// TIA Portal V18 export
FUNCTION_BLOCK "__mot_universal_"   // FB18, FBD
{ S7_Optimized_Access := 'TRUE' }
VERSION : 0.1
// stored: AutoNumber true, IsIECCheckEnabled false, IsRetainMemResEnabled false, MemoryReserve 100, SetENOAutomatically false, UDAEnableTagReadback false
   VAR_INPUT
      ALLOWED : Bool;
      ALLOWED_ONLY_IN_OVERRIDE : Bool;
      OVERRIDE_NOW : Bool;
      isMultiturn : Bool;
      MultiTurnGoesFwdOnly : Bool;
      xFwdOk : Bool;
      xRevOk : Bool;
      xPredefCal : Bool;
      MAN_SET_SPEED_maxParSpeed : Real;
      ENC : Real;
      par : "typeMotPara";
      partnerCalibrated : Bool := true;
      artLimits : Bool;
      artLimFwd : Real;
      artLimRev : Real;
      AU_EXECUTE_TO_TARGET : Bool;
      AU_SPD : Real;
      AUT_MD_SPD_notPos : Bool := false;
      AUT : Bool;
      MAN : Bool;
      CLOCK_S_P_SCAN { ExternalWritable := 'False'} : Real;
      ALIEN_HOST_CONTROL_MODE_ENABLE : Bool;
      ALIEN_FWD : Bool;
      ALIEN_REV : Bool;
      ALIEN_SPEED_ABS : Real;
      TheseAreDoors : Bool;
   END_VAR
   VAR_OUTPUT
      AU_INPOS : Bool;
      FWD : Bool;
      REV : Bool;
      BRK_REL : Bool;
      SPEED_ABS : Real;
      SPEED : Real;
      BLIND : Bool;
      ER_FOLLOW : Bool;
      ER_SET : Bool;
      ER_FWD : Bool;
      ER_REV : Bool;
      er_ws : WString;
   END_VAR
   VAR_IN_OUT
      AU_TRGT : Real;
      calibrated : Bool;
      POS : Real;
      ENC_RET_DATA : "typePOSMEMcalib";
   END_VAR
   VAR
      par_Local : "typeMotPara";
      SERV_block : Bool;
      AUTO_static : Bool;
      MAN_static : Bool := TRUE;
      M_MD { S7_SetPoint := 'True'} : "MD";
      ENC_DB { S7_SetPoint := 'True'} : "encoder";
      manual { S7_SetPoint := 'True'} : "manual_analog";
      auto { S7_SetPoint := 'True'} : "auto_analog_NORMAL";
      ENC_CHECK { S7_SetPoint := 'True'} : "enc_no_change_in_time";
      BRK_DB { S7_SetPoint := 'True'} : "BRK_FB";
      sr_auto { S7_SetPoint := 'True'} : "SR_TRIG";
      sr_man { S7_SetPoint := 'True'} : "SR_TRIG";
      auto_analog_Speed_Instance { S7_SetPoint := 'True'} : "auto_analog_copySpeed";
      speed_slowed_by_inertia : Real;
      speed_command : Real;
      mot_speed_wdir_slowly_accelerated_Instance { S7_SetPoint := 'True'} : "mot_speed_wdir_slowly_accelerated";
      mot_missed_target { S7_SetPoint := 'True'} : "mot_universal_arrived_missed";
      arrived_missed : Bool;
   END_VAR
   VAR_TEMP
      reset_y : Bool;
      BRK_NOW_ERROR_EXISTS : Bool;
      speed_fast_neg : Real;
      placeHolderreal : Real;
      er_set_1m : Bool;
      er_set_1a1 : Bool;
      er_set_1a2 : Bool;
      er_set_2 : Bool;
      er_set_3 : Bool;
      inertia_Mode : Bool;
      erws1m0 : WString;
      erws1a1 : WString;
      erws1a2 : WString;
      erws2 : WString;
      erws3 : WString;
   END_VAR
   VAR CONSTANT
      erwsNOER : WString := WSTRING#'no er';
   END_VAR
BEGIN

REGION Network 1
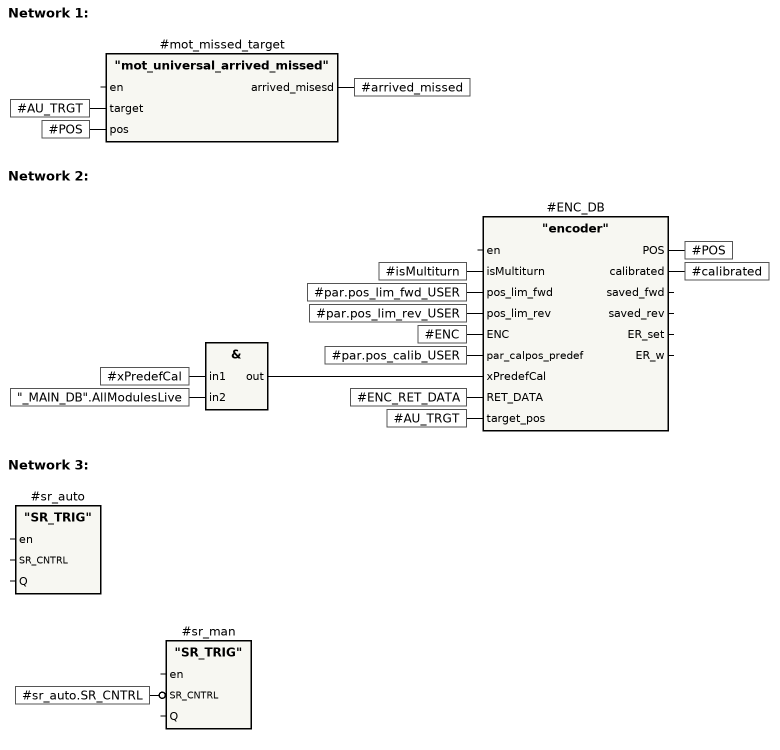
   #mot_missed_target(target := #AU_TRGT, pos := #POS, arrived_misesd => #arrived_missed);   // "mot_universal_arrived_missed"
END_REGION

REGION Network 2
   #ENC_DB(isMultiturn := #isMultiturn,   // "encoder"
           pos_lim_fwd := #par.pos_lim_fwd_USER,
           pos_lim_rev := #par.pos_lim_rev_USER,
           ENC := #ENC,
           par_calpos_predef := #par.pos_calib_USER,
           xPredefCal := #xPredefCal AND "_MAIN_DB".AllModulesLive,
           RET_DATA := #ENC_RET_DATA,
           target_pos := #AU_TRGT,
           POS => #POS,
           calibrated => #calibrated);
END_REGION

REGION Network 3
   #sr_auto();   // "SR_TRIG"
   #sr_man(SR_CNTRL := NOT #sr_auto.SR_CNTRL);   // "SR_TRIG"
END_REGION

REGION Network 4 (SCL)
   #SERV_block := #ALIEN_HOST_CONTROL_MODE_ENABLE;
   IF #SERV_block THEN
       #FWD := #ALIEN_FWD;
       #REV := #ALIEN_REV;
       #SPEED_ABS := #ALIEN_SPEED_ABS;
   END_IF;
END_REGION

REGION Network 5
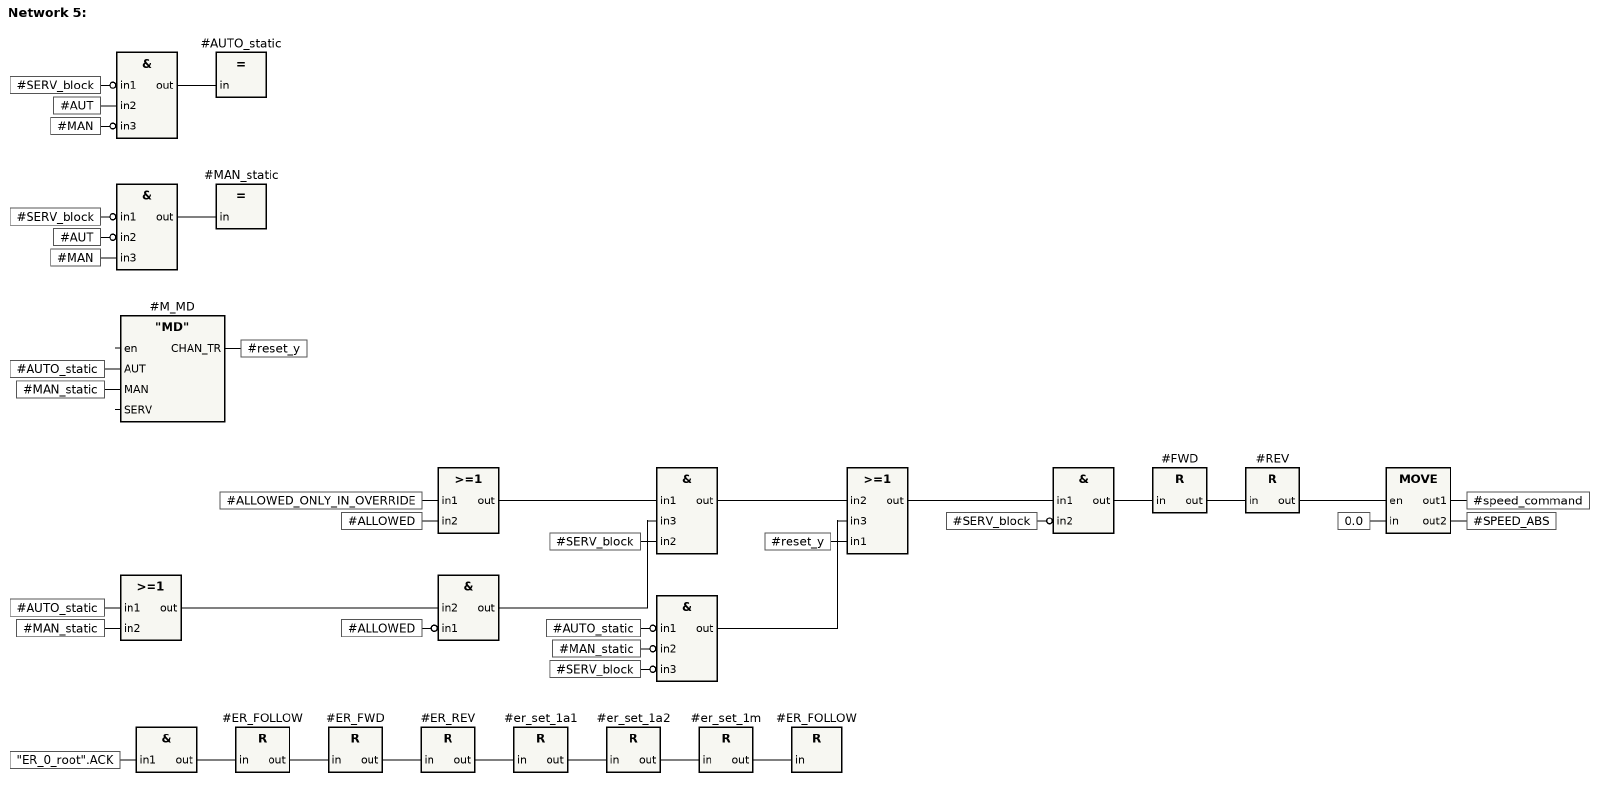
   #AUTO_static := NOT #SERV_block AND #AUT AND NOT #MAN;
   #MAN_static := NOT #SERV_block AND NOT #AUT AND #MAN;
   #M_MD(AUT := #AUTO_static, MAN := #MAN_static, CHAN_TR => #reset_y);   // "MD"
   IF (((#ALLOWED_ONLY_IN_OVERRIDE OR #ALLOWED) AND (#AUTO_static OR #MAN_static) AND NOT #ALLOWED AND #SERV_block) OR (NOT #AUTO_static AND NOT #MAN_static AND NOT #SERV_block) OR #reset_y) AND NOT #SERV_block THEN
       #FWD := FALSE;
       #REV := FALSE;
       #speed_command := 0.0;
       #SPEED_ABS := 0.0;
   END_IF;
   IF "ER_0_root".ACK THEN
       #ER_FOLLOW := FALSE;
       #ER_FWD := FALSE;
       #ER_REV := FALSE;
       #er_set_1a1 := FALSE;
       #er_set_1a2 := FALSE;
       #er_set_1m := FALSE;
       #ER_FOLLOW := FALSE;
   END_IF;
END_REGION

REGION Network 6
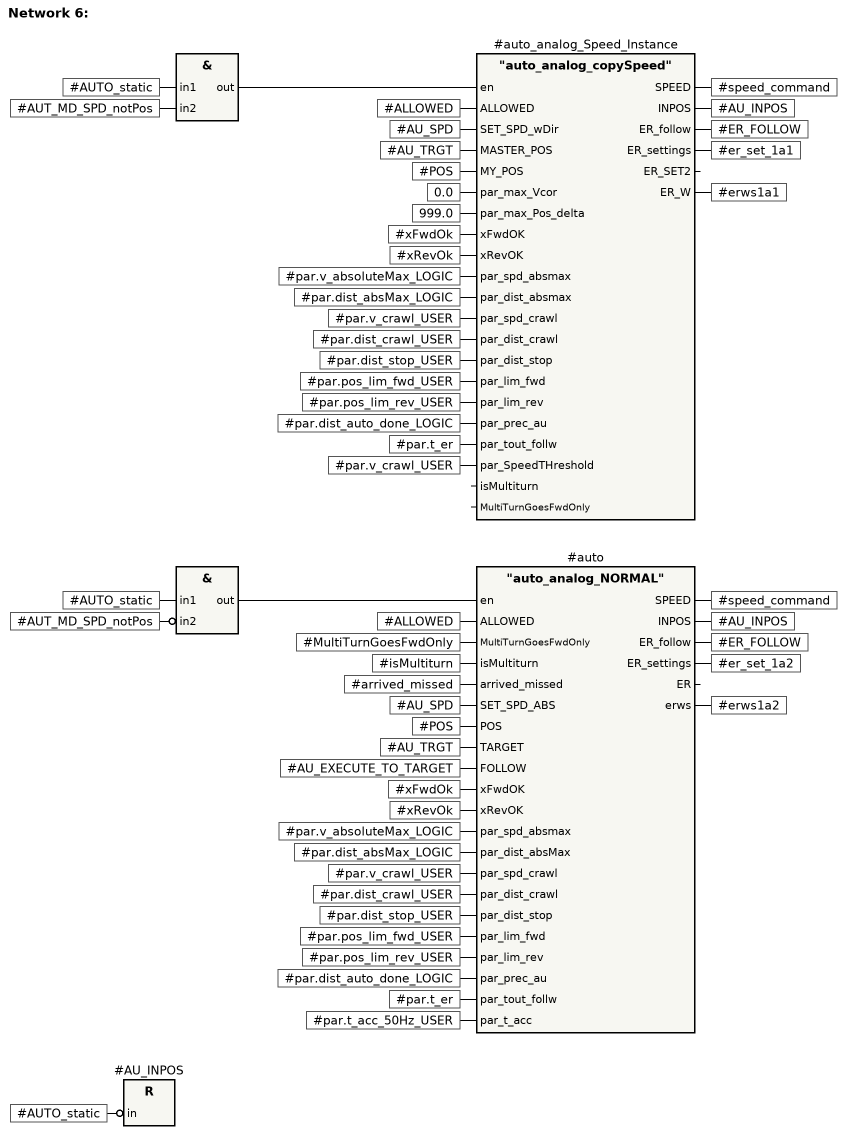
   IF #AUTO_static AND #AUT_MD_SPD_notPos THEN
       #auto_analog_Speed_Instance(ALLOWED := #ALLOWED,   // "auto_analog_copySpeed"
                               SET_SPD_wDir := #AU_SPD,
                               MASTER_POS := #AU_TRGT,
                               MY_POS := #POS,
                               par_max_Vcor := 0.0,
                               par_max_Pos_delta := 999.0,
                               xFwdOK := #xFwdOk,
                               xRevOK := #xRevOk,
                               par_spd_absmax := #par.v_absoluteMax_LOGIC,
                               par_dist_absmax := #par.dist_absMax_LOGIC,
                               par_spd_crawl := #par.v_crawl_USER,
                               par_dist_crawl := #par.dist_crawl_USER,
                               par_dist_stop := #par.dist_stop_USER,
                               par_lim_fwd := #par.pos_lim_fwd_USER,
                               par_lim_rev := #par.pos_lim_rev_USER,
                               par_prec_au := #par.dist_auto_done_LOGIC,
                               par_tout_follw := #par.t_er,
                               par_SpeedTHreshold := #par.v_crawl_USER,
                               SPEED => #speed_command,
                               INPOS => #AU_INPOS,
                               ER_follow => #ER_FOLLOW,
                               ER_settings => #er_set_1a1,
                               ER_W => #erws1a1);
   END_IF;
   IF #AUTO_static AND NOT #AUT_MD_SPD_notPos THEN
       #auto(ALLOWED := #ALLOWED,   // "auto_analog_NORMAL"
             MultiTurnGoesFwdOnly := #MultiTurnGoesFwdOnly,
             isMultiturn := #isMultiturn,
             arrived_missed := #arrived_missed,
             SET_SPD_ABS := #AU_SPD,
             POS := #POS,
             TARGET := #AU_TRGT,
             FOLLOW := #AU_EXECUTE_TO_TARGET,
             xFwdOK := #xFwdOk,
             xRevOK := #xRevOk,
             par_spd_absmax := #par.v_absoluteMax_LOGIC,
             par_dist_absMax := #par.dist_absMax_LOGIC,
             par_spd_crawl := #par.v_crawl_USER,
             par_dist_crawl := #par.dist_crawl_USER,
             par_dist_stop := #par.dist_stop_USER,
             par_lim_fwd := #par.pos_lim_fwd_USER,
             par_lim_rev := #par.pos_lim_rev_USER,
             par_prec_au := #par.dist_auto_done_LOGIC,
             par_tout_follw := #par.t_er,
             par_t_acc := #par.t_acc_50Hz_USER,
             SPEED => #speed_command,
             INPOS => #AU_INPOS,
             ER_follow => #ER_FOLLOW,
             ER_settings => #er_set_1a2,
             erws => #erws1a2);
   END_IF;
   IF NOT #AUTO_static THEN #AU_INPOS := FALSE; END_IF;
END_REGION

REGION Network 7 (SCL)

   //#MAN_SET_SPEED_maxParSpeed := #MAN_SET_SPEED_maxParSpeed;
END_REGION

REGION Network 8
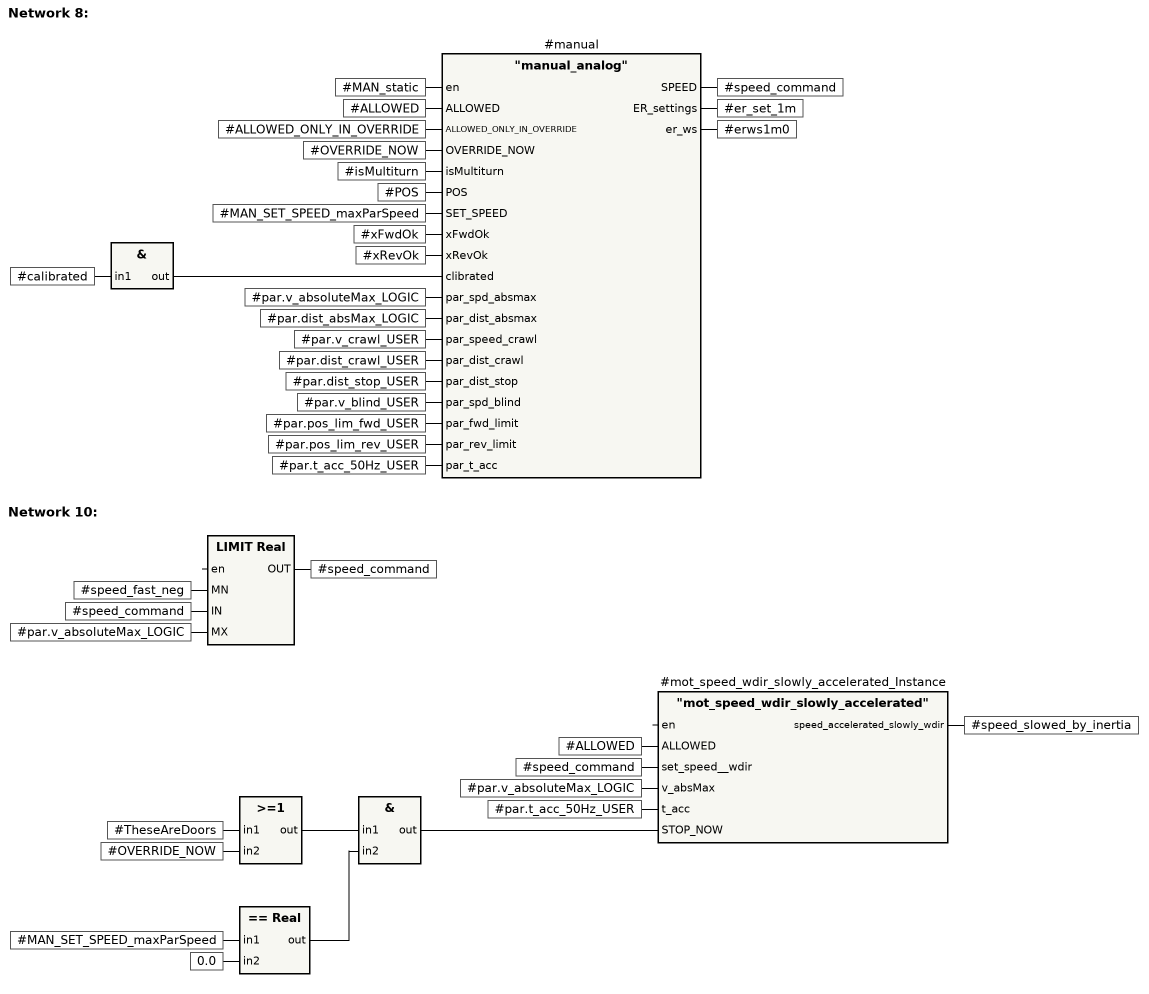
   IF #MAN_static THEN
       #manual(ALLOWED := #ALLOWED,   // "manual_analog"
               ALLOWED_ONLY_IN_OVERRIDE := #ALLOWED_ONLY_IN_OVERRIDE,
               OVERRIDE_NOW := #OVERRIDE_NOW,
               isMultiturn := #isMultiturn,
               POS := #POS,
               SET_SPEED := #MAN_SET_SPEED_maxParSpeed,
               xFwdOk := #xFwdOk,
               xRevOk := #xRevOk,
               clibrated := #calibrated,
               par_spd_absmax := #par.v_absoluteMax_LOGIC,
               par_dist_absmax := #par.dist_absMax_LOGIC,
               par_speed_crawl := #par.v_crawl_USER,
               par_dist_crawl := #par.dist_crawl_USER,
               par_dist_stop := #par.dist_stop_USER,
               par_spd_blind := #par.v_blind_USER,
               par_fwd_limit := #par.pos_lim_fwd_USER,
               par_rev_limit := #par.pos_lim_rev_USER,
               par_t_acc := #par.t_acc_50Hz_USER,
               SPEED => #speed_command,
               ER_settings => #er_set_1m,
               er_ws => #erws1m0);
   END_IF;
END_REGION

REGION Network 9 (SCL)
   #speed_fast_neg := -#par.v_absoluteMax_LOGIC;
END_REGION

REGION Network 10
   #speed_command := LIMIT(MN := #speed_fast_neg, IN := #speed_command, MX := #par.v_absoluteMax_LOGIC);
   #mot_speed_wdir_slowly_accelerated_Instance(ALLOWED := #ALLOWED,   // "mot_speed_wdir_slowly_accelerated"
                           set_speed__wdir := #speed_command,
                           v_absMax := #par.v_absoluteMax_LOGIC,
                           t_acc := #par.t_acc_50Hz_USER,
                           STOP_NOW := (#TheseAreDoors OR #OVERRIDE_NOW) AND (#MAN_SET_SPEED_maxParSpeed = 0.0),
                           speed_accelerated_slowly_wdir => #speed_slowed_by_inertia);
END_REGION

REGION Network 11 (SCL)
   IF NOT #SERV_block THEN
       #FWD := #speed_slowed_by_inertia > 0;
       #REV := #speed_slowed_by_inertia < 0;
   END_IF;
END_REGION

REGION Network 12
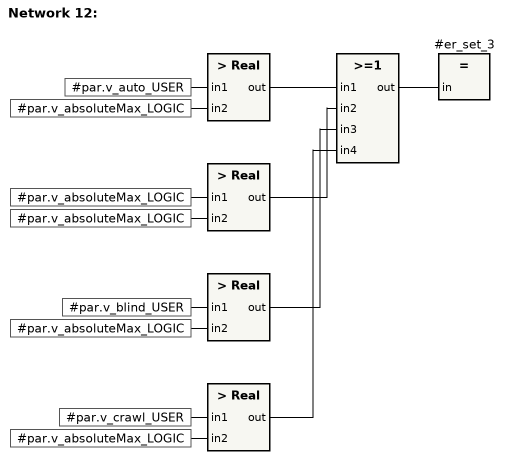
   #er_set_3 := (#par.v_auto_USER > #par.v_absoluteMax_LOGIC) OR (#par.v_absoluteMax_LOGIC > #par.v_absoluteMax_LOGIC) OR (#par.v_blind_USER > #par.v_absoluteMax_LOGIC) OR (#par.v_crawl_USER > #par.v_absoluteMax_LOGIC);
END_REGION

REGION Network 13
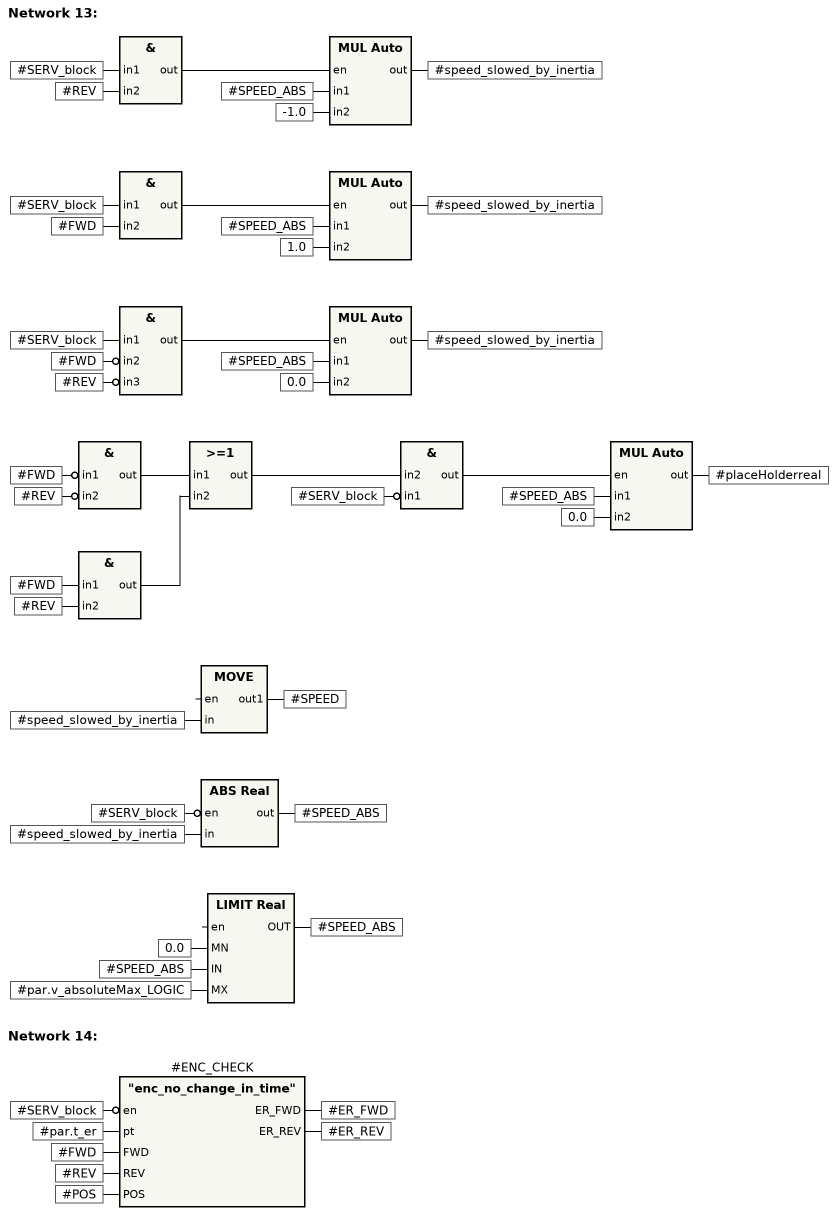
   IF #SERV_block AND #REV THEN #speed_slowed_by_inertia := #SPEED_ABS * (-1.0); END_IF;
   IF #SERV_block AND #FWD THEN #speed_slowed_by_inertia := #SPEED_ABS * 1.0; END_IF;
   IF #SERV_block AND NOT #FWD AND NOT #REV THEN #speed_slowed_by_inertia := #SPEED_ABS * 0.0; END_IF;
   IF ((NOT #FWD AND NOT #REV) OR (#FWD AND #REV)) AND NOT #SERV_block THEN
       #placeHolderreal := #SPEED_ABS * 0.0;
   END_IF;
   #SPEED := #speed_slowed_by_inertia;
   IF NOT #SERV_block THEN #SPEED_ABS := ABS(#speed_slowed_by_inertia); END_IF;
   #SPEED_ABS := LIMIT(MN := 0.0, IN := #SPEED_ABS, MX := #par.v_absoluteMax_LOGIC);
END_REGION

REGION Network 14
   IF NOT #SERV_block THEN
       #ENC_CHECK(pt := #par.t_er, FWD := #FWD, REV := #REV, POS := #POS, ER_FWD => #ER_FWD, ER_REV => #ER_REV);   // "enc_no_change_in_time"
   END_IF;
END_REGION

REGION Network 15
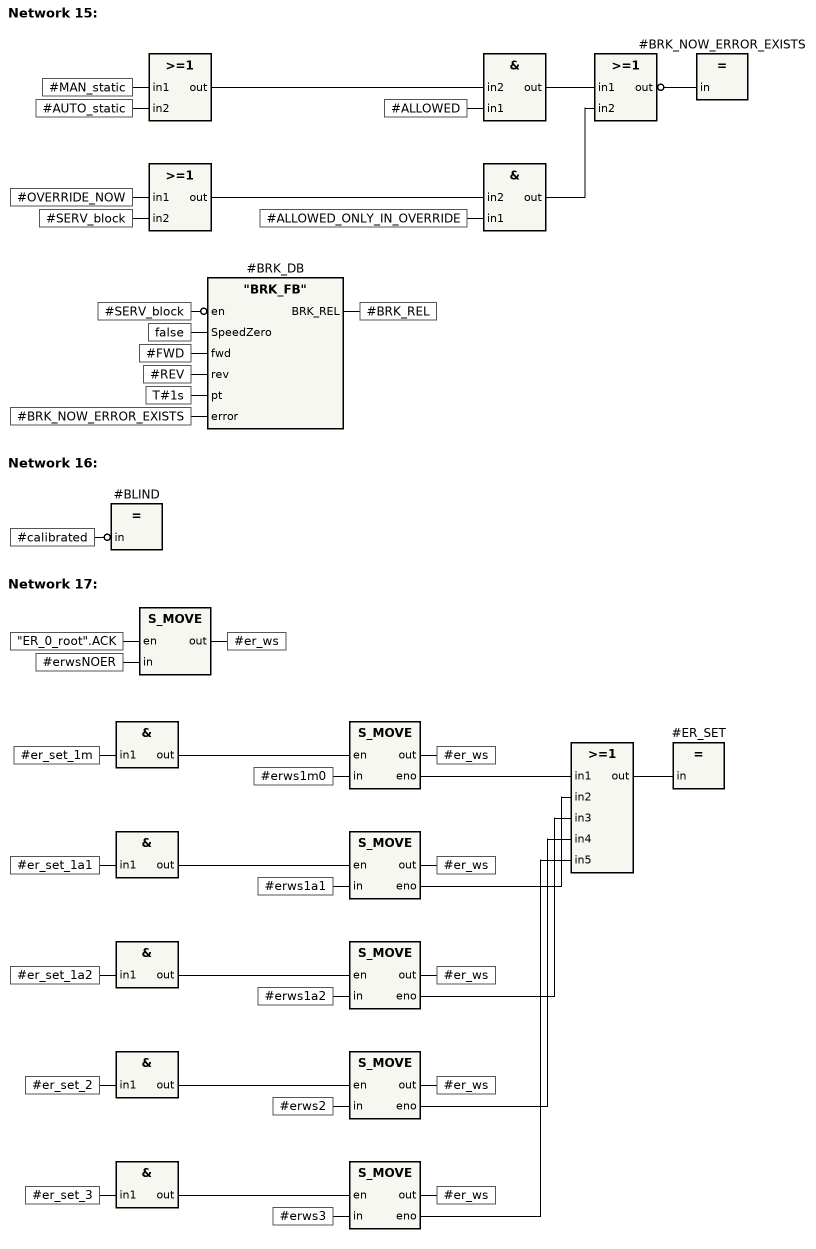
   #BRK_NOW_ERROR_EXISTS := NOT (((#MAN_static OR #AUTO_static) AND #ALLOWED) OR ((#OVERRIDE_NOW OR #SERV_block) AND #ALLOWED_ONLY_IN_OVERRIDE));
   IF NOT #SERV_block THEN
       #BRK_DB(SpeedZero := false,   // "BRK_FB"
               fwd := #FWD,
               rev := #REV,
               pt := T#1s,
               error := #BRK_NOW_ERROR_EXISTS,
               BRK_REL => #BRK_REL);
   END_IF;
END_REGION

REGION Network 16
   #BLIND := NOT #calibrated;
END_REGION

REGION Network 17
   IF "ER_0_root".ACK THEN #er_ws := #erwsNOER; END_IF;
   IF #er_set_1m THEN #er_ws := #erws1m0; END_IF;
   IF #er_set_1a1 THEN #er_ws := #erws1a1; END_IF;
   IF #er_set_1a2 THEN #er_ws := #erws1a2; END_IF;
   IF #er_set_2 THEN #er_ws := #erws2; END_IF;
   IF #er_set_3 THEN #er_ws := #erws3; END_IF;
   #ER_SET := #er_set_1m OR #er_set_1a1 OR #er_set_1a2 OR #er_set_2 OR #er_set_3;
END_REGION
END_FUNCTION_BLOCK
